FUNCTION_BLOCK PtDateTime IMPLEMENTS I_PtDateTime
VAR_INPUT
END_VAR
VAR_OUTPUT
END_VAR
VAR
	_Year : DINT;
	_Month : DINT;
	_Day : DINT;
	_Hour : DINT;
	_Minute : DINT;
	_Second : DINT;
	_Microsecond : DINT;
	_TimeZone : DINT;
	
END_VAR

PROPERTY Day : DINT
GET
Day := _Day;
END_GET
SET
_Day := Day;
END_SET
END_PROPERTY

METHOD Diff : I_PtInterval
VAR_INPUT
	TargetDateTime : PtDateTime;
END_VAR
//Diff.Set(THIS^,TargetDateTime,TRUE);
Pendulum._interval.Set(THIS^,TargetDateTime,TRUE);
Diff := Pendulum._interval;
END_METHOD

PROPERTY Hour : DINT
GET
Hour := _Hour;
END_GET
SET
_Hour := Hour;
END_SET
END_PROPERTY

PROPERTY Microsecond : DINT
GET
Microsecond := _Microsecond;
END_GET
SET
_Microsecond := Microsecond;
END_SET
END_PROPERTY

PROPERTY Minute : DINT
GET
Minute := _Minute;
END_GET
SET
_Minute := Minute;
END_SET
END_PROPERTY

PROPERTY Month : DINT
GET
Month := _Month;
END_GET
SET
_Month := Month;
END_SET
END_PROPERTY

PROPERTY Second : DINT
GET
Second := _Second;
END_GET
SET
_Second := Second;
END_SET
END_PROPERTY

METHOD Set //: PtDateTime
VAR_INPUT
	Year : DINT;
	Month : DINT;
	Day : DINT;
	Hour : DINT;
	Minute : DINT;
	Second : DINT;
	Microsecond : DINT;
	TimeZone : DINT;
END_VAR
THIS^._Year := Year;
THIS^._Month := Month;
THIS^._Day := Day;
THIS^._Hour := Hour;
THIS^._Minute := Minute;
THIS^._Second := Second;
THIS^._Microsecond := Microsecond;
THIS^._TimeZone := TimeZone;
END_METHOD

PROPERTY TimeZone : DINT
GET
TimeZone := _TimeZone;
END_GET
SET
_TimeZone := TimeZone;
END_SET
END_PROPERTY

PROPERTY Year : DINT
GET
Year := _Year;
END_GET
SET
_Year := Year;
END_SET
END_PROPERTY

END_FUNCTION_BLOCK

(* stored: Version 1.1.0.1, ProductVersion 3.1.4024.12
   POU PtDateTime: Id {199ef190-0e3e-494f-b841-5664fe8530fb}, SpecialFunc None
   Property Day: Id {83ae12ad-4977-4444-9a64-cae7ae009df5}
   Get Get: Id {b4ed34fa-4a29-4d3c-9ef8-45cc6d86184f}
   Set Set: Id {95bfc776-3013-4da9-9ae2-23d8b9727899}
   Method Diff: Id {43836bbc-fb61-416b-a2fb-80519b684688}
   Property Hour: Id {6d654241-0a93-4763-ab2e-ad9eabf843c9}
   Get Get: Id {f1e5a0a8-483a-42e9-8a1a-c0d909b9a6b4}
   Set Set: Id {51c66ded-a14d-4193-91f7-430353f4f74f}
   Property Microsecond: Id {470dfab1-3f0d-46ac-a7d5-dd500fae4ccb}
   Get Get: Id {7ab02b90-2238-436b-82b2-356b9aef50bf}
   Set Set: Id {e2fea909-453f-4cff-9a1d-70503d16fb18}
   Property Minute: Id {c4050bef-cfc3-4f6d-9468-5785b837dc13}
   Get Get: Id {60d0bc62-c136-4362-9a4b-33a419e357cf}
   Set Set: Id {e54273ae-738e-4cf8-8cf2-c605bb069e33}
   Property Month: Id {da181a09-6a77-44fd-97d6-64ae24d9353e}
   Get Get: Id {6bdfd857-332d-45b4-8cf6-7d6cac114c6f}
   Set Set: Id {eb61c076-e2c2-41a2-bf2c-37f6da51456e}
   Property Second: Id {dc7068b6-a80d-4287-ba96-cc8c2a285616}
   Get Get: Id {13b9c056-1fce-4415-b50e-4d43e30131f6}
   Set Set: Id {012e74b5-edda-4779-bf70-b8f6f2ef28de}
   Method Set: Id {7b7eb91f-ee8c-4fe0-b470-d2c2e4ca9f4e}
   Property TimeZone: Id {8e64c43b-80a6-4c8f-ac74-25474a461785}
   Get Get: Id {1b3469ca-610e-4ce8-a4ef-9a888bade90a}
   Set Set: Id {6bf9725d-7dd5-4975-9e54-471bcda973f6}
   Property Year: Id {020436fd-557d-45f9-8c9c-d71c4b4d9a12}
   Get Get: Id {f4b76565-a237-472d-98c4-299c5523480a}
   Set Set: Id {9fe522e8-5a9f-4d3b-85c9-6b841a7eb5a5} *)
